Staubli VAL3: TestSoap.dtx

mdesc mNomSpeed
jointRx jPos[2]
num nNum[2]
public pointRx pPos[2]
  [0] = {fatherId=world[0]}
  [1] = {fatherId=world[0]}
string sString
trsf trTrsf
frame fFrame = {fatherId=world[0]}
